// Implicitly generated code : DO NOT EDIT
FUNCTION CheckRangeSigned : DINT
VAR_INPUT
	value, lower, upper: DINT;
END_VAR

// Implicitly generated code : Only an Implementation suggestion
{noflow}
IF (value < lower) THEN
	CheckRangeSigned := lower;
	G_Diag.uiCheckRange:=G_Diag.uiCheckRange+1;
ELSIF(value > upper) THEN
	CheckRangeSigned := upper;
	G_Diag.uiCheckRange:=G_Diag.uiCheckRange+1;
ELSE
	CheckRangeSigned := value;
END_IF
{flow}

END_FUNCTION

(* stored: Version 1.1.0.1, ProductVersion 3.1.4024.4
   POU CheckRangeSigned: Id {e7072a03-b9be-4a65-94a8-3dca0a5c41e8}, SpecialFunc CheckRangeSigned *)
